GLOBALCONSTANTS byteconst (* Global constants *)
  (* Standard: 61499-1 *)
  (* Version 1.0, 2024-02-22, franz *)
  VAR_GLOBAL CONSTANT
    WORD_BYTE_ZZ : WORD := 16#0000; (* ZERO Constant *)
    SHFT_BYTE_00 : SINT := 0; (* shift 0 bits *)
    WORD_BYTE_00 : WORD := 16#00FF; (* LSB_Byte Constant *)
    SHFT_BYTE_01 : SINT := 8; (* shift 8 bits *)
    WORD_BYTE_01 : WORD := 16#FF00; (* MSB_Byte Constant *)
  END_VAR
END_GLOBALCONSTANTS
